// TIA Portal V18 export
TYPE "UDT_DailyScheduler"
// stored: IsFailsafeCompliant false
   STRUCT
      Start : Time_Of_Day;
      Stop : Time_Of_Day;
   END_STRUCT;
END_TYPE
